INTERFACE I_HandoverListener

METHOD M_HandoverCompleteEvent
VAR_INPUT
END_VAR
END_METHOD

METHOD M_HandoverStartEvent
VAR_INPUT
END_VAR
END_METHOD

END_INTERFACE

(* stored: Version 1.1.0.1, ProductVersion 3.1.4022.12
   Itf I_HandoverListener: Id {1329ef7b-f0a9-45a6-9dda-e7dfc50fb37e}
   Method M_HandoverCompleteEvent: Id {7be36221-1f02-4a4d-b9ff-61384a829a59}
   Method M_HandoverStartEvent: Id {51fe2f8e-3e77-4e6e-bf3f-57913ac9a02c} *)
